{attribute 'global_init_slot' := '40500'} //https://infosys.beckhoff.com/index.php?content=../content/1031/tc3_plc_intro/2529649291.html&id=
VAR_GLOBAL CONSTANT
	MaxNrofMessages: UINT:= 30;
	emptySkill : FB_1_Skill; //emptySkill
END_VAR


{attribute 'global_init_slot' := '40600'} //https://infosys.beckhoff.com/index.php?content=../content/1031/tc3_plc_intro/2529649291.html&id=
//Skills
VAR_GLOBAL
	skPP: Skill_PickPlace := (
		sPickName:='P1',
		sPlaceName:='P2'
	);
	skEy: Skill_ROS2_Eyes;	

END_VAR


{attribute 'global_init_slot' := '40700'} //https://infosys.beckhoff.com/index.php?content=../content/1031/tc3_plc_intro/2529649291.html&id=
//Robots
VAR_GLOBAL
	// 	BFH_RobLab_UR5: ROBOT_UR5 :=(
// 		sRobotIp:='192.168.250.2',
// 		pA_Skills:= [ADR(skPP),ADR(skEy)]
// 	);
// 	BFH_RobLab_UR5e: ROBOT_UR5 :=(
// 		sRobotIp:='192.168.250.2',
// 		pA_Skills:= [ADR(skPP),ADR(skEy)]
// 	);

	ETA_Ausb_UR5: ROBOT_UR5 :=(
		sRobotIp:='192.168.250.2',
		pA_Skills:= [ADR(skPP),ADR(skEy)]
	);
	
// 	ETA_TechCenter_LD90: FB_OmronLD90;
// 	ETA_Meca500: FB_Meca500;
END_VAR


VAR_GLOBAL
// 	PLC: FB_0_Base;
END_VAR

(* stored: Version 1.1.0.1, ProductVersion 3.1.4026.18
   GVL SETUP: Id {c749aa94-77ca-4d45-832d-ac09e2bd2780} *)
